PROGRAM MAIN
VAR
END_VAR

END_PROGRAM

(* stored: Version 1.1.0.1
   POU MAIN: Id {a4fcd149-2d0c-46ea-a8b2-a0ae08469da4} *)
